// Mitsubishi GX Works2 project: test   PLC: FX3U/FX3UC

PROGRAM MAIN
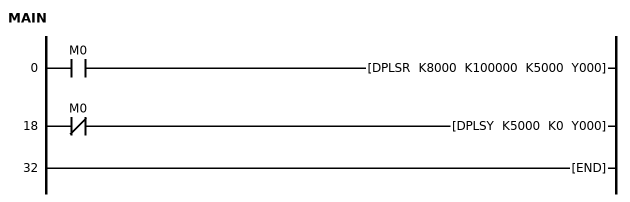
0     LD      M0
      DPLSR   K8000 K100000 K5000 Y000
18    LDI     M0
      DPLSY   K5000 K0 Y000
32    END
END_PROGRAM
